PROGRAM C10_PackControlOCVData
VAR
	aDisablePackAggregCamera	: ARRAY[1..3] OF BOOL;

	tonWriteLoopWatchog			: TON;
	rtWriteOCVFile					: R_TRIG;
	fbWriteOCVFileLoop			: FB_PACK_WriteOCVLoopDB;

	fbPackLevelCounter			: FB_KPI_PackLevelCounter;
	rtOCVValidation				: R_TRIG;

	aOCVDataCounters			: ARRAY[0..3] OF R_TRIG;

	fbFileWriteOCVError			: FB_LOG_FileWriteError;
END_VAR

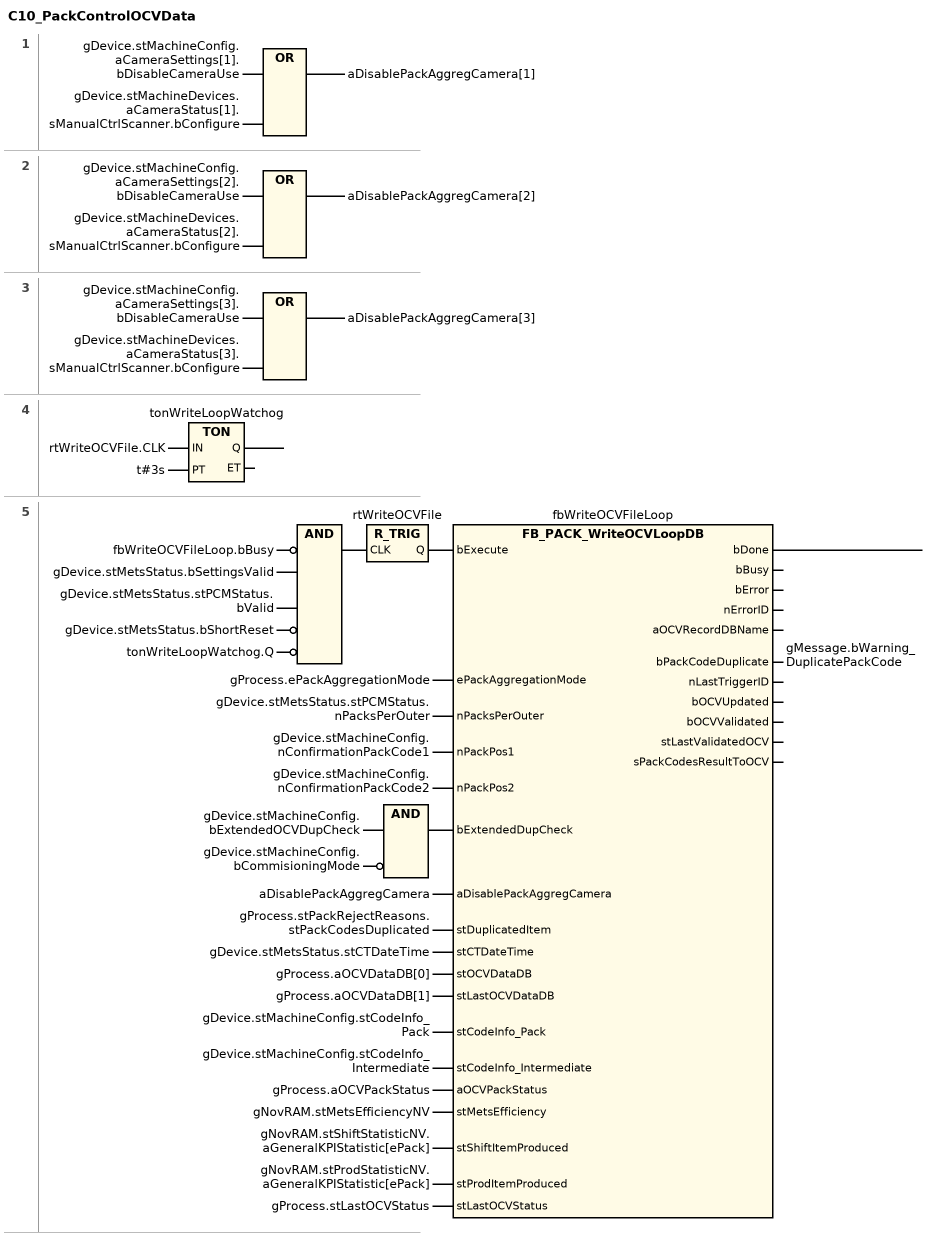
// NETWORK 1
aDisablePackAggregCamera[1] := gDevice.stMachineConfig.aCameraSettings[1].bDisableCameraUse OR gDevice.stMachineDevices.aCameraStatus[1].sManualCtrlScanner.bConfigure;

// NETWORK 2
aDisablePackAggregCamera[2] := gDevice.stMachineConfig.aCameraSettings[2].bDisableCameraUse OR gDevice.stMachineDevices.aCameraStatus[2].sManualCtrlScanner.bConfigure;

// NETWORK 3
aDisablePackAggregCamera[3] := gDevice.stMachineConfig.aCameraSettings[3].bDisableCameraUse OR gDevice.stMachineDevices.aCameraStatus[3].sManualCtrlScanner.bConfigure;

// NETWORK 4
tonWriteLoopWatchog(IN := rtWriteOCVFile.CLK, PT := t#3s); // TON

// NETWORK 5
rtWriteOCVFile(CLK := NOT fbWriteOCVFileLoop.bBusy AND gDevice.stMetsStatus.bSettingsValid AND gDevice.stMetsStatus.stPCMStatus.bValid AND NOT gDevice.stMetsStatus.bShortReset AND NOT tonWriteLoopWatchog.Q); // R_TRIG
fbWriteOCVFileLoop(
    bExecute := rtWriteOCVFile.Q,
    ePackAggregationMode := gProcess.ePackAggregationMode,
    nPacksPerOuter := gDevice.stMetsStatus.stPCMStatus.nPacksPerOuter,
    nPackPos1 := gDevice.stMachineConfig.nConfirmationPackCode1,
    nPackPos2 := gDevice.stMachineConfig.nConfirmationPackCode2,
    bExtendedDupCheck := gDevice.stMachineConfig.bExtendedOCVDupCheck AND NOT gDevice.stMachineConfig.bCommisioningMode,
    aDisablePackAggregCamera := aDisablePackAggregCamera,
    stDuplicatedItem := gProcess.stPackRejectReasons.stPackCodesDuplicated,
    stCTDateTime := gDevice.stMetsStatus.stCTDateTime,
    stOCVDataDB := gProcess.aOCVDataDB[0],
    stLastOCVDataDB := gProcess.aOCVDataDB[1],
    stCodeInfo_Pack := gDevice.stMachineConfig.stCodeInfo_Pack,
    stCodeInfo_Intermediate := gDevice.stMachineConfig.stCodeInfo_Intermediate,
    aOCVPackStatus := gProcess.aOCVPackStatus,
    stMetsEfficiency := gNovRAM.stMetsEfficiencyNV,
    stShiftItemProduced := gNovRAM.stShiftStatisticNV.aGeneralKPIStatistic[ePack],
    stProdItemProduced := gNovRAM.stProdStatisticNV.aGeneralKPIStatistic[ePack],
    stLastOCVStatus := gProcess.stLastOCVStatus,
    bPackCodeDuplicate => gMessage.bWarning_DuplicatePackCode); // FB_PACK_WriteOCVLoopDB

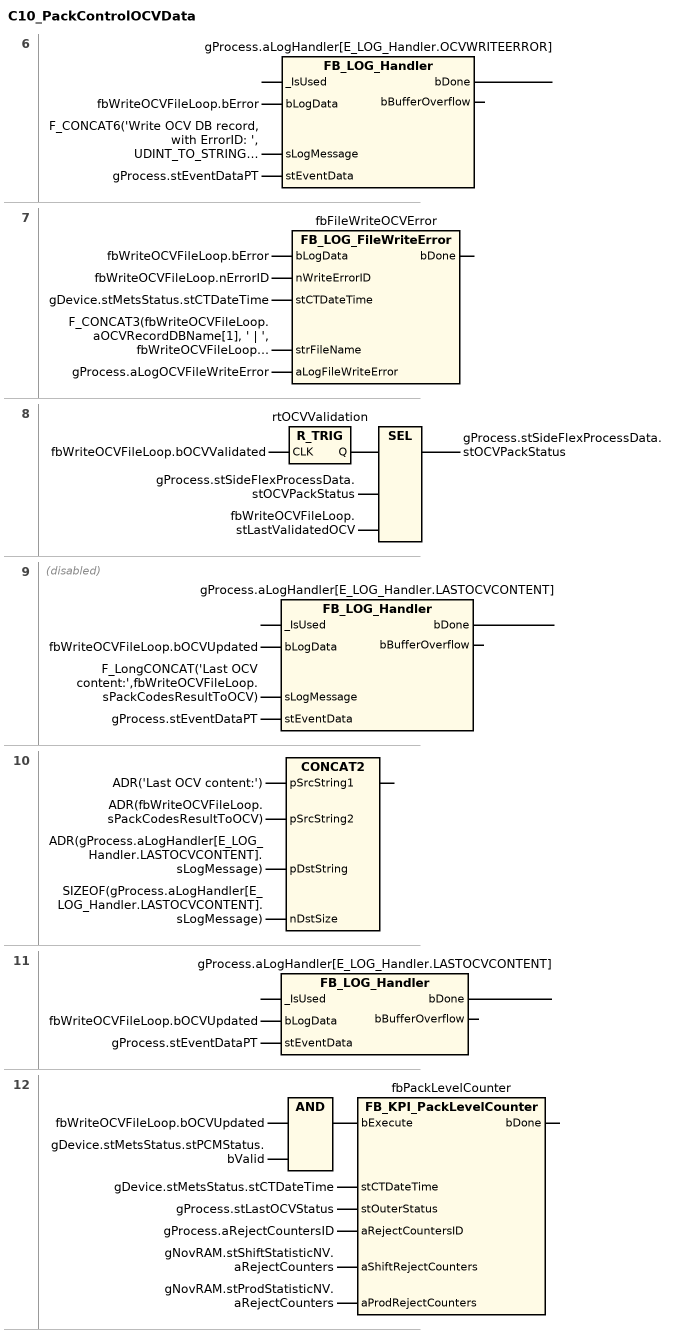
// NETWORK 6
gProcess.aLogHandler[E_LOG_Handler.OCVWRITEERROR](
    bLogData := fbWriteOCVFileLoop.bError,
    sLogMessage := F_CONCAT6('Write OCV DB record, with ErrorID: ', UDINT_TO_STRING(fbWriteOCVFileLoop.nErrorID), '. OCV 1: ', fbWriteOCVFileLoop.aOCVRecordDBName[1],  '. OCV 2: ', fbWriteOCVFileLoop.aOCVRecordDBName[2]),
    stEventData := gProcess.stEventDataPT); // FB_LOG_Handler

// NETWORK 7
fbFileWriteOCVError(
    bLogData := fbWriteOCVFileLoop.bError,
    nWriteErrorID := fbWriteOCVFileLoop.nErrorID,
    stCTDateTime := gDevice.stMetsStatus.stCTDateTime,
    strFileName := F_CONCAT3(fbWriteOCVFileLoop.aOCVRecordDBName[1], ' | ', fbWriteOCVFileLoop.aOCVRecordDBName[2]),
    aLogFileWriteError := gProcess.aLogOCVFileWriteError); // FB_LOG_FileWriteError

// NETWORK 8
rtOCVValidation(CLK := fbWriteOCVFileLoop.bOCVValidated); // R_TRIG
gProcess.stSideFlexProcessData.stOCVPackStatus := SEL(rtOCVValidation.Q, gProcess.stSideFlexProcessData.stOCVPackStatus, fbWriteOCVFileLoop.stLastValidatedOCV);

// NETWORK 9 (disabled)
// gProcess.aLogHandler[E_LOG_Handler.LASTOCVCONTENT](
//     bLogData := fbWriteOCVFileLoop.bOCVUpdated,
//     sLogMessage := F_LongCONCAT('Last OCV content:',fbWriteOCVFileLoop.sPackCodesResultToOCV),
//     stEventData := gProcess.stEventDataPT); // FB_LOG_Handler

// NETWORK 10
CONCAT2(pSrcString1 := ADR('Last OCV content:'), pSrcString2 := ADR(fbWriteOCVFileLoop.sPackCodesResultToOCV), pDstString := ADR(gProcess.aLogHandler[E_LOG_Handler.LASTOCVCONTENT].sLogMessage), nDstSize := SIZEOF(gProcess.aLogHandler[E_LOG_Handler.LASTOCVCONTENT].sLogMessage));

// NETWORK 11
gProcess.aLogHandler[E_LOG_Handler.LASTOCVCONTENT](bLogData := fbWriteOCVFileLoop.bOCVUpdated, stEventData := gProcess.stEventDataPT); // FB_LOG_Handler

// NETWORK 12
fbPackLevelCounter(
    bExecute := fbWriteOCVFileLoop.bOCVUpdated AND gDevice.stMetsStatus.stPCMStatus.bValid,
    stCTDateTime := gDevice.stMetsStatus.stCTDateTime,
    stOuterStatus := gProcess.stLastOCVStatus,
    aRejectCountersID := gProcess.aRejectCountersID,
    aShiftRejectCounters := gNovRAM.stShiftStatisticNV.aRejectCounters,
    aProdRejectCounters := gNovRAM.stProdStatisticNV.aRejectCounters); // FB_KPI_PackLevelCounter

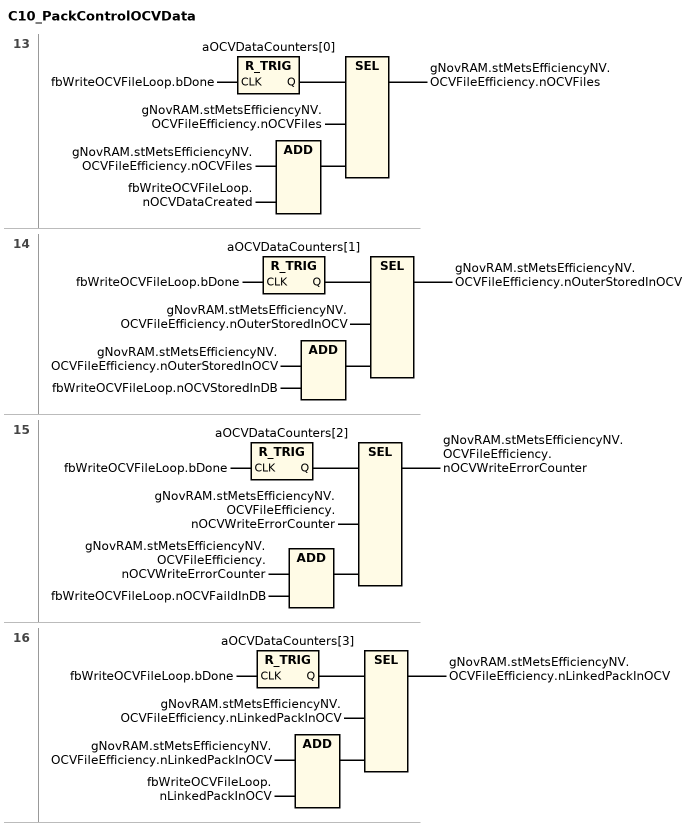
// NETWORK 13
aOCVDataCounters[0](CLK := fbWriteOCVFileLoop.bDone); // R_TRIG
gNovRAM.stMetsEfficiencyNV.OCVFileEfficiency.nOCVFiles := SEL(aOCVDataCounters[0].Q, gNovRAM.stMetsEfficiencyNV.OCVFileEfficiency.nOCVFiles, gNovRAM.stMetsEfficiencyNV.OCVFileEfficiency.nOCVFiles + fbWriteOCVFileLoop.nOCVDataCreated);

// NETWORK 14
aOCVDataCounters[1](CLK := fbWriteOCVFileLoop.bDone); // R_TRIG
gNovRAM.stMetsEfficiencyNV.OCVFileEfficiency.nOuterStoredInOCV := SEL(aOCVDataCounters[1].Q, gNovRAM.stMetsEfficiencyNV.OCVFileEfficiency.nOuterStoredInOCV, gNovRAM.stMetsEfficiencyNV.OCVFileEfficiency.nOuterStoredInOCV + fbWriteOCVFileLoop.nOCVStoredInDB);

// NETWORK 15
aOCVDataCounters[2](CLK := fbWriteOCVFileLoop.bDone); // R_TRIG
gNovRAM.stMetsEfficiencyNV.OCVFileEfficiency.nOCVWriteErrorCounter := SEL(aOCVDataCounters[2].Q, gNovRAM.stMetsEfficiencyNV.OCVFileEfficiency.nOCVWriteErrorCounter, gNovRAM.stMetsEfficiencyNV.OCVFileEfficiency.nOCVWriteErrorCounter + fbWriteOCVFileLoop.nOCVFaildInDB);

// NETWORK 16
aOCVDataCounters[3](CLK := fbWriteOCVFileLoop.bDone); // R_TRIG
gNovRAM.stMetsEfficiencyNV.OCVFileEfficiency.nLinkedPackInOCV := SEL(aOCVDataCounters[3].Q, gNovRAM.stMetsEfficiencyNV.OCVFileEfficiency.nLinkedPackInOCV, gNovRAM.stMetsEfficiencyNV.OCVFileEfficiency.nLinkedPackInOCV + fbWriteOCVFileLoop.nLinkedPackInOCV);

END_PROGRAM

(* stored: Version 1.1.0.1
   POU C10_PackControlOCVData: Id {0a216cd4-197c-48a2-9eca-7da4b3c7e299}, SpecialFunc None *)
